(* IEC 61131-3 sources: T4Exjobb/Sigma/Stations/Terminal/HMI/Class/_SyncTimeHMI, 1 file *)

(* ---- _SyncTimeHMI.st ---- *)
(*!
<Class
	Name               = "_SyncTimeHMI"
	Revision           = "2.0"
	RealtimeTask       = "false"
	CyclicTask         = "false"
	BackgroundTask     = "true"
	DefBackground      = "100 ms"
	Sigmatek           = "true"
	OSInterface        = "false"
	HighPriority       = "false"
	Automatic          = "false"
	UpdateMode         = "Prescan"
	SharedCommandTable = "true"
	Objectsize         = "(540,180)"
	Comment            = "class reads date and time from two clients (within the adjusted zycletime)&#13;&#10;and writes these values to the servers">
	<Channels>
		<Server Name="sSyncDate" Visualized="true" Initialize="false" WriteProtected="false" Retentive="false" Comment="server for sync date - also input is possible"/>
		<Server Name="sSyncTime" Visualized="true" Initialize="false" WriteProtected="false" Retentive="false" Comment="server for sync time - also input is possible"/>
		<Client Name="ActDate" Required="true" Internal="false" Comment="actual date"/>
		<Client Name="ActTime" Required="true" Internal="false" Comment="actual time"/>
		<Client Name="SetDate" Required="false" Internal="false" Comment="destination date (e.g. for Machine Control)"/>
		<Client Name="SetTime" Required="false" Internal="false" Comment="destination time (e.g. for Machine Control)"/>
	</Channels>
	<Dependencies>
		<Files>
			<File Path=".\Class\_SyncTimeHMI\_SyncTimeHMI_de.pdf"/>
			<File Path=".\Class\_SyncTimeHMI\_SyncTimeHMI_en.pdf"/>
		</Files>
	</Dependencies>
	<RevDoku>
		<Owner Company="Sigmatek"/>
		<Dokumentation Revision="2.0" Date="2018-02-07" Author="KaiAnd" Company="Sigmatek" Description="Implemented functionality to take over date &amp; time of inputs on server vars&#13;&#10;--&gt; server for date &amp; time now have write() mwthods for inputs&#13;&#10;--&gt; new destination clients SetDate and SetTime (optional)"/>
		<Dokumentation Revision="1.1" Date="2016-10-10" Author="HubChr" Company="Sigmatek" Description="Added documentation pdfs."/>
		<Dokumentation Revision="1.0" Date="2015-11-11" Author="hötant" Company="Sigmatek" Description="creation of class"/>
	</RevDoku>
</Class>
*)
_SyncTimeHMI : CLASS
  //Servers:
	sSyncDate 	: SvrChCmd_DATE_LSL;
	sSyncTime 	: SvrCh_TIME_LSL;
  //Clients:
	ActDate 	: CltCh_HDINT;
	ActTime 	: CltCh_HDINT;
	SetDate 	: CltCh_HDINT;
	SetTime 	: CltCh_HDINT;
  //Variables:
		IsCon_SetDate 	: DINT;			//! <Variable Comment="&quot;Is Connected&quot; flag ..." Name="IsCon_SetDate"/>
		IsCon_SetTime 	: DINT;			//! <Variable Comment="&quot;Is Connected&quot; flag ..." Name="IsCon_SetTime"/>
		TimeStampSync 	: UDINT;
  //Functions:

	FUNCTION VIRTUAL GLOBAL Init;

	FUNCTION VIRTUAL GLOBAL Background
		VAR_INPUT
			EAX 	: UDINT;
		END_VAR
		VAR_OUTPUT
			state (EAX) 	: UDINT;
		END_VAR;

	FUNCTION VIRTUAL GLOBAL sSyncDate::Read
		VAR_OUTPUT
			output (EAX) 	: DATE_LSL;
		END_VAR;

	FUNCTION VIRTUAL GLOBAL sSyncDate::Write
		VAR_INPUT
			input (EAX) 	: DATE_LSL;
		END_VAR
		VAR_OUTPUT
			result (EAX) 	: DATE_LSL;
		END_VAR;

	FUNCTION VIRTUAL GLOBAL sSyncTime::Read
		VAR_OUTPUT
			output (EAX) 	: TIME_LSL;
		END_VAR;

	FUNCTION VIRTUAL GLOBAL sSyncTime::Write
		VAR_INPUT
			input (EAX) 	: TIME_LSL;
		END_VAR
		VAR_OUTPUT
			result (EAX) 	: TIME_LSL;
		END_VAR;
  //Tables:
	FUNCTION @STD
		VAR_OUTPUT
			ret_code	: CONFSTATES;
		END_VAR;
	FUNCTION GLOBAL TAB @CT_;
END_CLASS;

FUNCTION VIRTUAL GLOBAL _SyncTimeHMI::Init

  if (_FirstScan) then

    //-------------------------------------------------------------------------
    //  check client-connnections and set flags                         V.2.0
    //-------------------------------------------------------------------------
    IsCon_SetDate := FALSE;
    IsCon_SetTime := FALSE;
    if (IsClientConnected(#SetDate)) then   IsCon_SetDate := TRUE; end_if;
    if (IsClientConnected(#SetTime)) then   IsCon_SetTime := TRUE; end_if;
    //-------------------------------------------------------------------------

  end_if;

END_FUNCTION

FUNCTION VIRTUAL GLOBAL _SyncTimeHMI::Background
	VAR_INPUT
		EAX 	: UDINT;
	END_VAR
	VAR_OUTPUT
		state (EAX) 	: UDINT;
	END_VAR

	state := READY;

  //---------------------------------------------------------------------------
  //  TimeSync without inputs on sSync-servers ... V.2.0
  //---------------------------------------------------------------------------
  ActDate := ActDate.Read();
  ActTime := ActTime.Read();

  if ((ops.tAbsolute - TimeStampSync) >= 20000) then
    TimeStampSync := ops.tAbsolute;

    if (IsCon_SetDate = TRUE) then
      SetDate := ActDate ;
      SetDate.Write(ActDate);
    end_if;

    if (IsCon_SetTime = TRUE) then
      SetTime := ActTime ;
      SetTime.Write(ActTime);
    end_if;

  end_if;
  //---------------------------------------------------------------------------

END_FUNCTION

FUNCTION VIRTUAL GLOBAL _SyncTimeHMI::sSyncDate::Read
	VAR_OUTPUT
		output (EAX) 	: DATE_LSL;
	END_VAR

 output := sSyncDate := ActDate := ActDate.Read();

END_FUNCTION

FUNCTION VIRTUAL GLOBAL _SyncTimeHMI::sSyncTime::Read
	VAR_OUTPUT
		output (EAX) 	: TIME_LSL;
	END_VAR

	output := sSyncTime := ActTime := ActTime.Read();

END_FUNCTION

FUNCTION VIRTUAL GLOBAL _SyncTimeHMI::sSyncDate::Write
	VAR_INPUT
		input (EAX) 	: DATE_LSL;
	END_VAR
	VAR_OUTPUT
		result (EAX) 	: DATE_LSL;
	END_VAR

	sSyncDate := input;
	result := sSyncDate;

  // write input date to destination
  ActDate := sSyncDate ;
  ActDate.Write(sSyncDate);

  if (IsCon_SetDate = TRUE) then
    SetDate := sSyncDate ;
    SetDate.Write(sSyncDate);
  end_if;

END_FUNCTION

FUNCTION VIRTUAL GLOBAL _SyncTimeHMI::sSyncTime::Write
	VAR_INPUT
		input (EAX) 	: TIME_LSL;
	END_VAR
	VAR_OUTPUT
		result (EAX) 	: TIME_LSL;
	END_VAR

	sSyncTime := input;
	result := sSyncTime;

  // write input time to destination
  ActTime := sSyncTime ;
  ActTime.Write(sSyncTime);

  if (IsCon_SetTime = TRUE) then
    SetTime := sSyncTime ;
    SetTime.Write(sSyncTime);
  end_if;

END_FUNCTION
